Yaskawa INFORM job: POS-DATA.JBI

/JOB
//NAME POS-DATA
//POS
///NPOS 0,0,0,8,0,0
///TOOL 0
///POSTYPE PULSE
///PULSE
P00000=4209,-7192,-5593,1580,-64891,83596
P00010=59507,31722,-17078,218,-38821,63431
P00011=-57751,18396,-30102,118,-37151,107094
P00012=-57751,4620,-10147,94,-56535,107123
P00013=-62194,-3771,-4505,-26,-60500,-580
P00014=-62194,-3771,13695,-26,-5676,-580
P00015=56762,19251,10333,925,-63692,64135
P00016=56762,19251,10333,925,-63692,64135
//INST
///DATE 2024/08/21 18:16
///ATTR SC,RW
///GROUP1 RB1
NOP
*1
IFTHENEXP IN#(6)=ON
	 SET B010 1
	 SET B011 2
	 SET B012 3
	 MOVJ P000 VJ=I002
	 MOVJ P[B010] VJ=I002
	 SET I010 11
	 MOVJ P[B011] VJ=I003
	 DOUT OT#(2) ON
	 SET I010 12
	 MOVL P[B012] V=I003
	 DOUT OT#(1) ON
	 TIMER T=1.000
	 SET I010 11
	 MOVL P[B011] V=I003
	 MOVJ P[B010] VJ=I002
	 MOVJ P000 VJ=I002
	 DOUT OT#(2) OFF
	 DOUT OT#(1) OFF
	 CLEAR I010 ALL
ENDIF
IFTHENEXP IN#(7)=ON
	 SET B010 4
	 SET B011 5
	 SET B012 6
	 MOVJ P000 VJ=I002
	 MOVJ P[B010] VJ=I002
	 SET I011 11
	 MOVJ P[B011] VJ=I003
	 DOUT OT#(4) ON
	 SET I011 12
	 MOVL P[B012] V=I003
	 DOUT OT#(3) ON
	 TIMER T=1.000
	 SET I011 11
	 MOVL P[B011] V=I003
	 MOVJ P[B010] VJ=I002
	 MOVJ P000 VJ=I002
	 DOUT OT#(4) OFF
	 DOUT OT#(3) OFF
	 CLEAR I011 ALL
ENDIF
COMM IFTHENEXP IN#(6)=OFF ANDEXP IN#(7)=OFF
COMM 	 MOVJ P010 VJ=15.00
COMM 	 MOVJ P011 VJ=15.00
COMM 	 MOVJ P012 VJ=15.00
COMM 	 MOVJ P013 VJ=15.00
COMM 	 MOVJ P014 VJ=15.00
COMM 	 MOVJ P015 VJ=15.00
COMM 	 MOVJ P016 VJ=15.00
COMM 	 MOVJ P000 VJ=15.00
COMM ENDIF
JUMP *1
END
